FUNCTION_BLOCK TUnitTestUnderTest EXTENDS TUnitTestBase
VAR_INPUT
END_VAR
VAR_OUTPUT
END_VAR
VAR
END_VAR

END_FUNCTION_BLOCK

(* stored: Version 1.1.0.1, ProductVersion 3.1.4024.4
   POU TUnitTestUnderTest: Id {7bfed642-dce0-402f-827d-e5704a2c4489}, SpecialFunc None *)
